(* Logix 5000 project; controller Drives_Line1 1756-L72 rev 20.13; software revision 20.04; part 12 of 21 *)
(* tags used below, declared in another part *)
   Bridle_02 : UDT_Bridle_2M;
   Bridle_03 : UDT_Bridle_2M;
   cu : UDT_Pinchroll;
   In_Commands : UDT_Commands;
   LineCmd : UDT_Commands_Line;
   LineCtrl : UDT_Control_Line;
   Out_Feedbacks : UDT_Fdbks;
   Out_Status : UDT_Status;
   TaskInterval_ms : DINT;
   TestConfig_Bridle_02a : UDT_Config_Bridle;
   TestConfig_Bridle_02b : UDT_Config_Bridle;
   TestConfig_cu : UDT_Config_Pinch;
   zConfigFromMaster : BOOL;
   zCuSpdTrimMltp : REAL;
   zPi : REAL;
   zSimulation : BOOL;
(* P15_Bridle_02, continued *)

ROUTINE R98_ToDrive   (* ladder *)
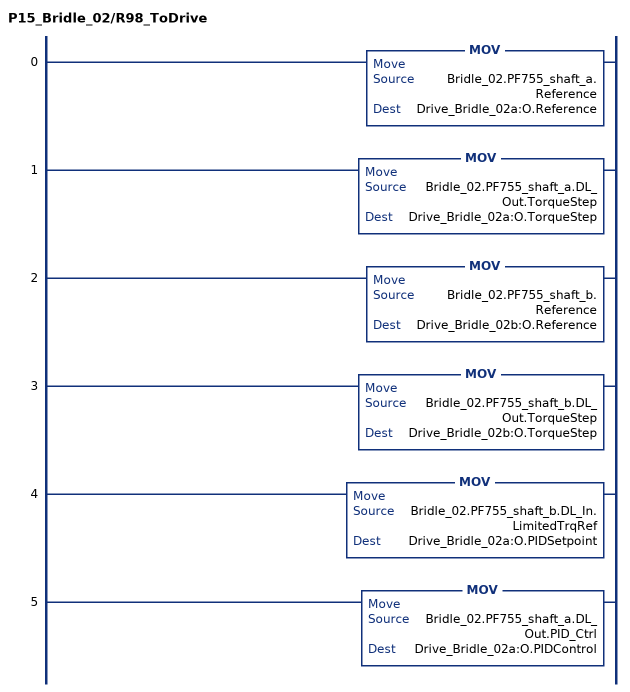
   0: MOV(Bridle_02.PF755_shaft_a.Reference,Drive_Bridle_02a:O.Reference);
   1: MOV(Bridle_02.PF755_shaft_a.DL_Out.TorqueStep,Drive_Bridle_02a:O.TorqueStep);
   2: MOV(Bridle_02.PF755_shaft_b.Reference,Drive_Bridle_02b:O.Reference);
   3: MOV(Bridle_02.PF755_shaft_b.DL_Out.TorqueStep,Drive_Bridle_02b:O.TorqueStep);
   4: MOV(Bridle_02.PF755_shaft_b.DL_In.LimitedTrqRef,Drive_Bridle_02a:O.PIDSetpoint);
   5: MOV(Bridle_02.PF755_shaft_a.DL_Out.PID_Ctrl,Drive_Bridle_02a:O.PIDControl);
END_ROUTINE

ROUTINE R999_Test   (* ladder *)
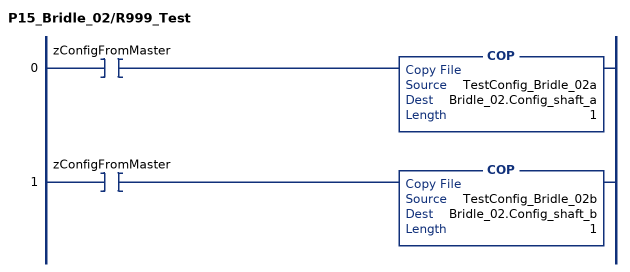
   0: XIC(zConfigFromMaster)COP(TestConfig_Bridle_02a,Bridle_02.Config_shaft_a,1);
   1: XIC(zConfigFromMaster)COP(TestConfig_Bridle_02b,Bridle_02.Config_shaft_b,1);
END_ROUTINE

ROUTINE R99_To_Master   (* ladder *)
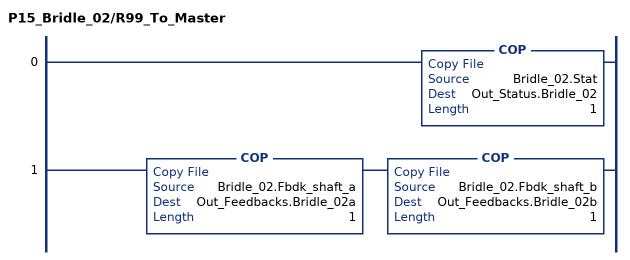
   0: COP(Bridle_02.Stat,Out_Status.Bridle_02,1);
   1: COP(Bridle_02.Fbdk_shaft_a,Out_Feedbacks.Bridle_02a,1)COP(Bridle_02.Fbdk_shaft_b,Out_Feedbacks.Bridle_02b,1);
END_ROUTINE
END_PROGRAM

PROGRAM P15b_rl_Cu   (* main routine R00_Main *)
VAR
   ADD_01 : FBD_MATH := (SourceB := 0.00068994303, Dest := 0.00068994303);
   aux1 : REAL;
   aux2 : REAL;
   BAND_01 : FBD_BOOLEAN_AND := (In3 := 1, In4 := 1, In5 := 1, In6 := 1, In7 := 1, In8 := 1);
   BAND_03 : FBD_BOOLEAN_AND := (In3 := 1, In4 := 1, In5 := 1, In6 := 1, In7 := 1, In8 := 1);
   BNOT_01 : FBD_BOOLEAN_NOT := (In := 1);
   BNOT_04 : FBD_BOOLEAN_NOT := (Out := 1);
   BNOT_06 : FBD_BOOLEAN_NOT := (Out := 1);
   cu2_Max_FBcounts : REAL := 5120.0;
   cu_FB_Count_Old : DINT;
   cu_FB_Diff : DINT;
   cu_FB_Update_Valid : BOOL;
   cu_Max_FBcounts : REAL := 5120.0;
   cu_RPMPerMPS : REAL := 5512.139;
   cu_SpdTrimMPS : REAL := 3.1769214e-06;
   cu_SpdTrimPct : REAL := 0.032127563;
   DIV_01 : FBD_MATH := (SourceA := 0.00053545943, SourceB := 100.0, Dest := 5.354594e-06);
   EQU_01 : FBD_COMPARE := (SourceA := 0.083333336);
   IO_State_cu : INT := 4;
   IO_State_Tmp_cu : INT := 16384;
   MUL_01 : FBD_MATH := (SourceA := 0.00068994303, SourceB := 5512.139, Dest := 3.803062);
   MUL_02 : FBD_MATH := (SourceA := 0.2);
   MUL_05 : FBD_MATH := (SourceA := 0.049963027, SourceB := 0.016666668, Dest := 0.00083271717);
   NEG_04 : FBD_MATH_ADVANCED := (Source := 0.233, Dest := -0.233);
   Ons : DINT := 1;
   PI_02 : PROP_INT := (In := 0.0045986176, Kp := 0.8, Wld := 0.1, HighLimit := 2.5, LowLimit := -2.5, ShapeKpPlus := 1.0, ShapeKpMinus := 1.0, ShapeWldPlus := 1.0, ShapeWldMinus := 1.0, RTSTime := 1, Out := 0.033255614, DeltaT := 0.05);
   PulsReset_PID : TIMER := (PRE := 250);
   RLIM_01 : RATE_LIMITER := (In := 0.00068994303, IncRate := 0.5, DecRate := 0.5, RTSTime := 1, Out := 0.00068994303, DeltaT := 0.05);
   SCL_09 : SCALE := (In := 0.1839509, InRawMax := 100.0, InRawMin := -100.0, InEUMax := 2.5, InEUMin := -2.5, Limiting := 1, Out := 0.0045986176);
   SCRV_01 : S_CURVE := (Initialize := 1, AbsAlgRamp := 1, AccelRate := 0.16, DecelRate := 0.16, JerkRate := 0.25, RTSTime := 1, DeltaT := 0.05);
   SSUM_03 : SELECTED_SUMMER := (In1 := 0.233, Gain1 := 1.0, In2 := -0.233, Gain2 := 1.0, Gain3 := 1.0, Select3 := 1, Gain4 := 1.0, Gain5 := 1.0, Gain6 := 1.0, Gain7 := 1.0, Gain8 := 1.0);
   SSUM_05 : SELECTED_SUMMER := (In1 := 0.00068994303, Gain1 := 1.0, Select1 := 1, Gain2 := 1.0, Gain3 := 1.0, Gain4 := 1.0, Gain5 := 1.0, Gain6 := 1.0, Gain7 := 1.0, Gain8 := 1.0, Out := 0.00068994303);
   SUB_02 : FBD_MATH := (SourceA := 6.741889, SourceB := 6.6660895, Dest := 0.075799465);
   TimeOn_PIDOn : TIMER := (PRE := 500);
   TofReset : TIMER := (PRE := 1000, ACC := 1000);
   TonNoResponse : TIMER[3] := ([0].PRE := 2500, [1].PRE := 2500, [2].PRE := 2500, [2].ACC := 2500, [2].EN := 1, [2].DN := 1);
   TonRefOn : TIMER := (PRE := 500);
   zcu_EncRes : DINT := 4096;
   zcu_Ki_SpdTrim : REAL := 0.1;
   zcu_Kp_SpdTrim : REAL := 0.8;
   zcu_Max_rev : DINT := 1500;
   zcu_MaxAccDec : REAL := 0.5;
   zcu_MaxTrimSpdTrim : REAL := 2.5;
   zcu_MinTrimSpdTrim : REAL := -2.5;
END_VAR

ROUTINE R00_Main   (* ladder *)
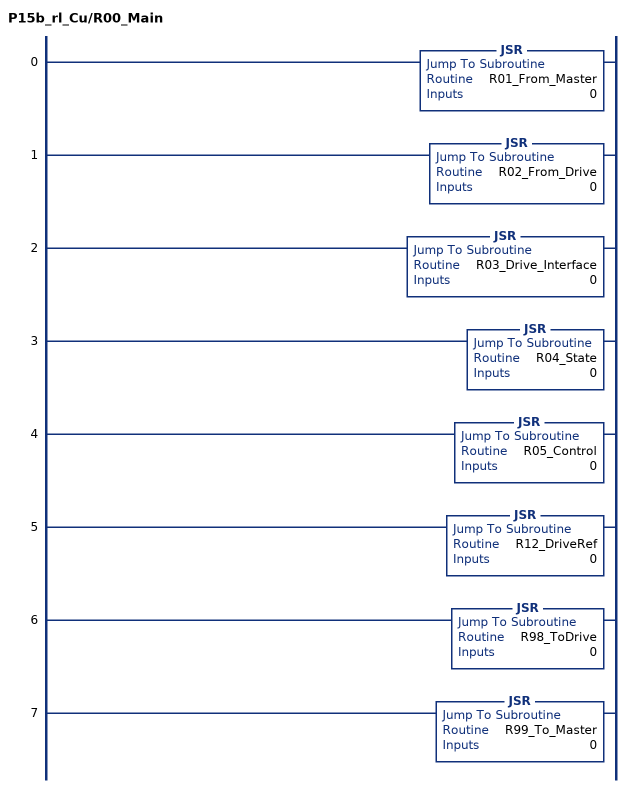
   0: JSR(R01_From_Master,0);
   1: JSR(R02_From_Drive,0);
   2: JSR(R03_Drive_Interface,0);
   3: JSR(R04_State,0);
   4: JSR(R05_Control,0);
   5: JSR(R12_DriveRef,0);
   6: JSR(R98_ToDrive,0);
   7: JSR(R99_To_Master,0);
END_ROUTINE

ROUTINE R01_From_Master   (* ladder *)
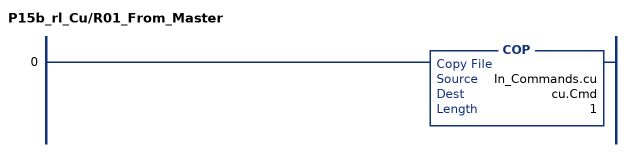
   0: COP(In_Commands.cu,cu.Cmd,1);
END_ROUTINE

ROUTINE R02_From_Drive   (* ladder *)
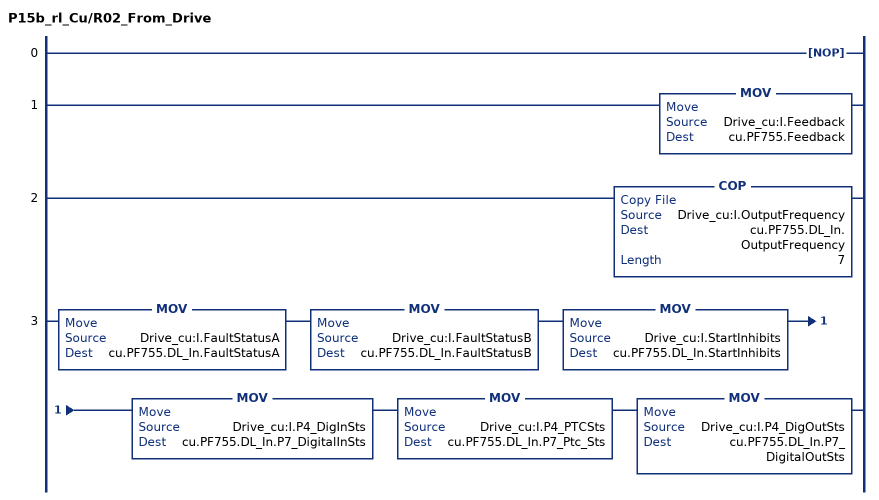
   0: NOP();
   1: MOV(Drive_cu:I.Feedback,cu.PF755.Feedback);
   2: COP(Drive_cu:I.OutputFrequency,cu.PF755.DL_In.OutputFrequency,7);
   3: MOV(Drive_cu:I.FaultStatusA,cu.PF755.DL_In.FaultStatusA)MOV(Drive_cu:I.FaultStatusB,cu.PF755.DL_In.FaultStatusB)MOV(Drive_cu:I.StartInhibits,cu.PF755.DL_In.StartInhibits)MOV(Drive_cu:I.P4_DigInSts,cu.PF755.DL_In.P7_DigitalInSts)MOV(Drive_cu:I.P4_PTCSts,cu.PF755.DL_In.P7_Ptc_Sts)MOV(Drive_cu:I.P4_DigOutSts,cu.PF755.DL_In.P7_DigitalOutSts);
END_ROUTINE

ROUTINE R03_Drive_Interface   (* ladder *)
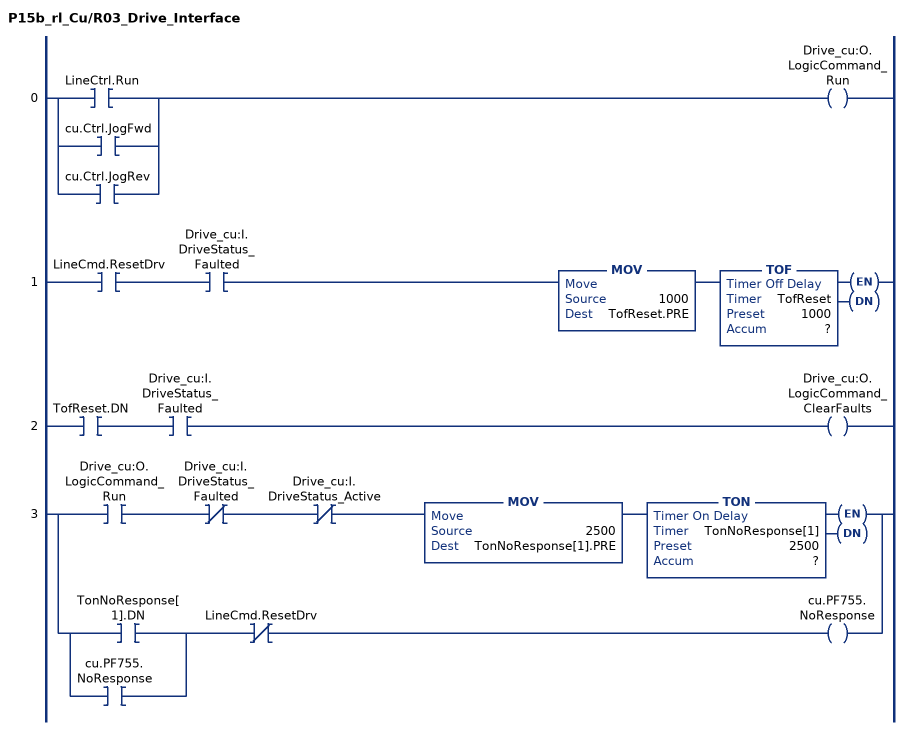
   0: [XIC(LineCtrl.Run) ,XIC(cu.Ctrl.JogFwd) ,XIC(cu.Ctrl.JogRev) ]OTE(Drive_cu:O.LogicCommand_Run);
   1: XIC(LineCmd.ResetDrv)XIC(Drive_cu:I.DriveStatus_Faulted)MOV(1000,TofReset.PRE)TOF(TofReset,?,?);
   2: XIC(TofReset.DN)XIC(Drive_cu:I.DriveStatus_Faulted)OTE(Drive_cu:O.LogicCommand_ClearFaults);
   3: [XIC(Drive_cu:O.LogicCommand_Run) XIO(Drive_cu:I.DriveStatus_Faulted) XIO(Drive_cu:I.DriveStatus_Active) MOV(2500,TonNoResponse[1].PRE) TON(TonNoResponse[1],?,?) ,[XIC(TonNoResponse[1].DN) ,XIC(cu.PF755.NoResponse) ] XIO(LineCmd.ResetDrv) OTE(cu.PF755.NoResponse) ];
END_ROUTINE

ROUTINE R04_State   (* ladder *)
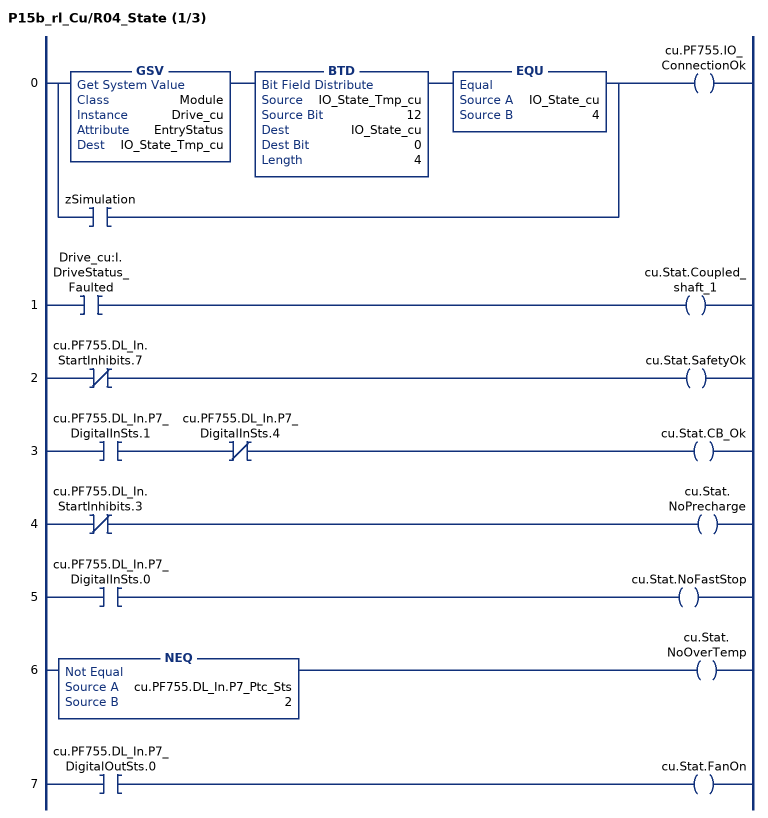
   0: [GSV(Module,Drive_cu,EntryStatus,IO_State_Tmp_cu) BTD(IO_State_Tmp_cu,12,IO_State_cu,0,4) EQU(IO_State_cu,4) ,XIC(zSimulation) ]OTE(cu.PF755.IO_ConnectionOk);
   1: XIC(Drive_cu:I.DriveStatus_Faulted)OTE(cu.Stat.Coupled_shaft_1);
   2: XIO(cu.PF755.DL_In.StartInhibits.7)OTE(cu.Stat.SafetyOk);
   3: XIC(cu.PF755.DL_In.P7_DigitalInSts.1)XIO(cu.PF755.DL_In.P7_DigitalInSts.4)OTE(cu.Stat.CB_Ok);
   4: XIO(cu.PF755.DL_In.StartInhibits.3)OTE(cu.Stat.NoPrecharge);
   5: XIC(cu.PF755.DL_In.P7_DigitalInSts.0)OTE(cu.Stat.NoFastStop);
   6: NEQ(cu.PF755.DL_In.P7_Ptc_Sts,2)OTE(cu.Stat.NoOverTemp);
   7: XIC(cu.PF755.DL_In.P7_DigitalOutSts.0)OTE(cu.Stat.FanOn);
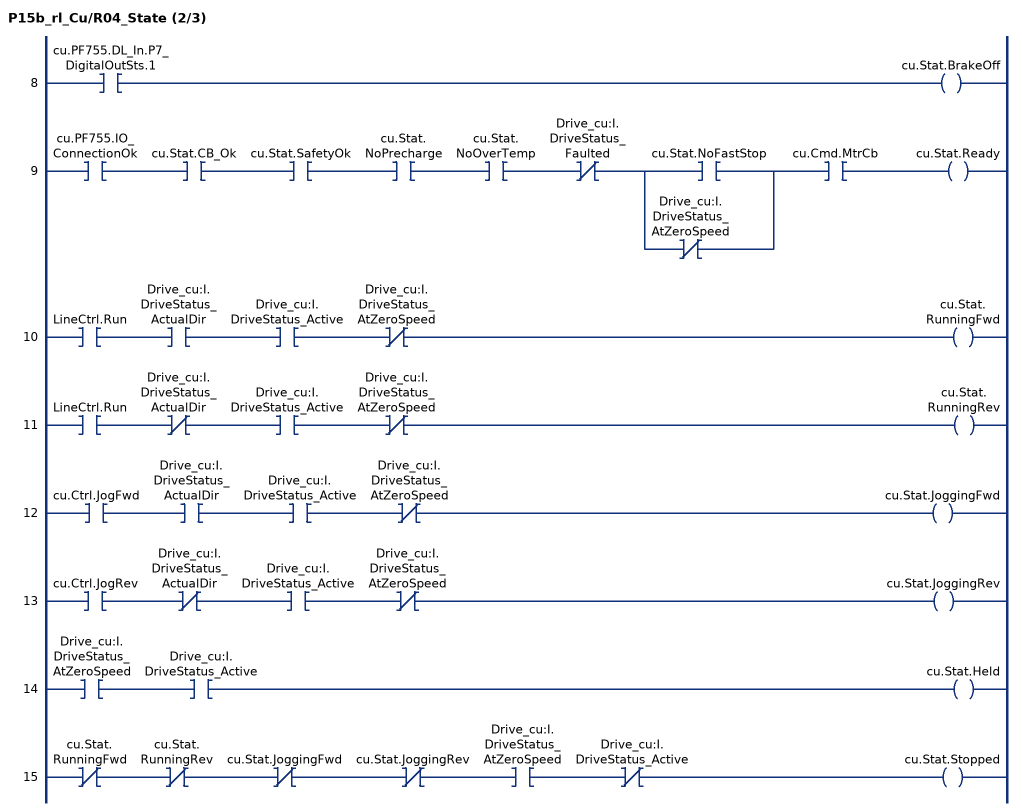
   8: XIC(cu.PF755.DL_In.P7_DigitalOutSts.1)OTE(cu.Stat.BrakeOff);
   9: XIC(cu.PF755.IO_ConnectionOk)XIC(cu.Stat.CB_Ok)XIC(cu.Stat.SafetyOk)XIC(cu.Stat.NoPrecharge)XIC(cu.Stat.NoOverTemp)XIO(Drive_cu:I.DriveStatus_Faulted)[XIC(cu.Stat.NoFastStop) ,XIO(Drive_cu:I.DriveStatus_AtZeroSpeed) ]XIC(cu.Cmd.MtrCb)OTE(cu.Stat.Ready);
   10: XIC(LineCtrl.Run)XIC(Drive_cu:I.DriveStatus_ActualDir)XIC(Drive_cu:I.DriveStatus_Active)XIO(Drive_cu:I.DriveStatus_AtZeroSpeed)OTE(cu.Stat.RunningFwd);
   11: XIC(LineCtrl.Run)XIO(Drive_cu:I.DriveStatus_ActualDir)XIC(Drive_cu:I.DriveStatus_Active)XIO(Drive_cu:I.DriveStatus_AtZeroSpeed)OTE(cu.Stat.RunningRev);
   12: XIC(cu.Ctrl.JogFwd)XIC(Drive_cu:I.DriveStatus_ActualDir)XIC(Drive_cu:I.DriveStatus_Active)XIO(Drive_cu:I.DriveStatus_AtZeroSpeed)OTE(cu.Stat.JoggingFwd);
   13: XIC(cu.Ctrl.JogRev)XIO(Drive_cu:I.DriveStatus_ActualDir)XIC(Drive_cu:I.DriveStatus_Active)XIO(Drive_cu:I.DriveStatus_AtZeroSpeed)OTE(cu.Stat.JoggingRev);
   14: XIC(Drive_cu:I.DriveStatus_AtZeroSpeed)XIC(Drive_cu:I.DriveStatus_Active)OTE(cu.Stat.Held);
   15: XIO(cu.Stat.RunningFwd)XIO(cu.Stat.RunningRev)XIO(cu.Stat.JoggingFwd)XIO(cu.Stat.JoggingRev)XIC(Drive_cu:I.DriveStatus_AtZeroSpeed)XIO(Drive_cu:I.DriveStatus_Active)OTE(cu.Stat.Stopped);
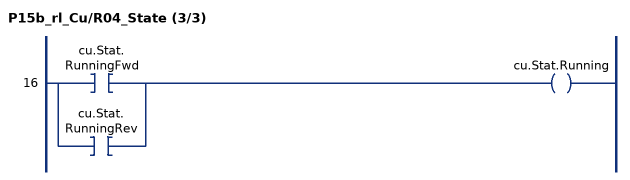
   16: [XIC(cu.Stat.RunningFwd) ,XIC(cu.Stat.RunningRev) ]OTE(cu.Stat.Running);
END_ROUTINE

ROUTINE R05_Control   (* ladder *)
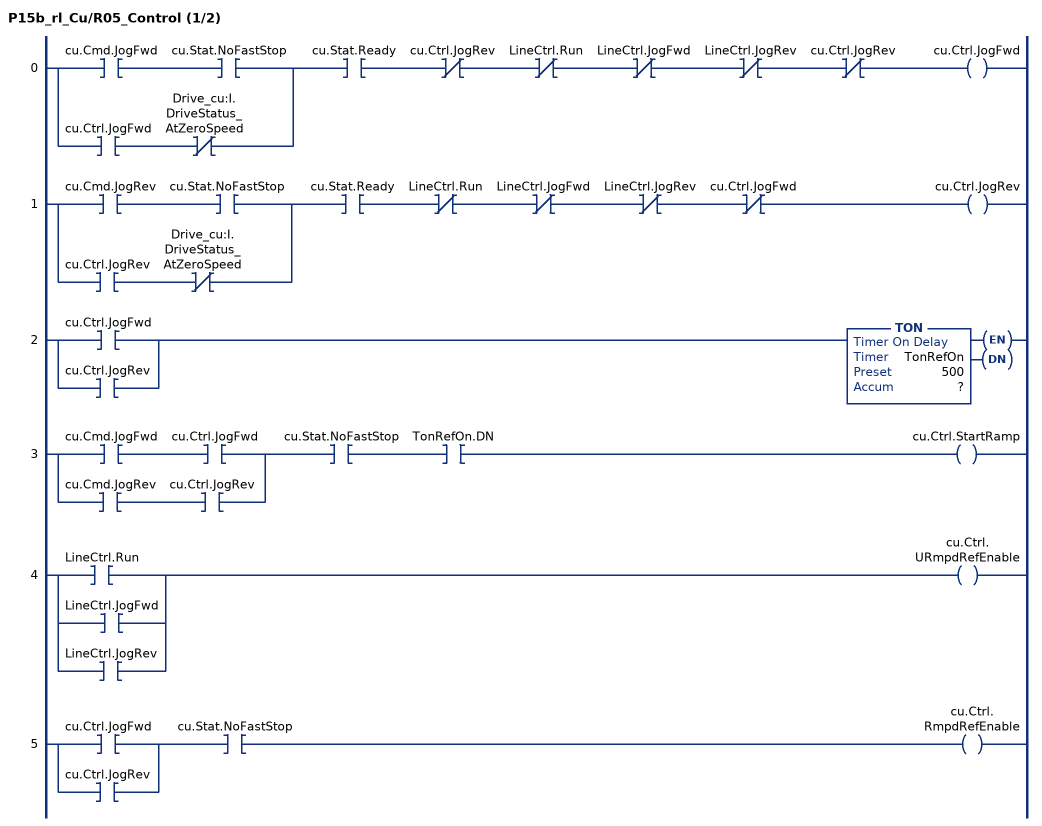
   0: [XIC(cu.Cmd.JogFwd) XIC(cu.Stat.NoFastStop) ,XIC(cu.Ctrl.JogFwd) XIO(Drive_cu:I.DriveStatus_AtZeroSpeed) ]XIC(cu.Stat.Ready)XIO(cu.Ctrl.JogRev)XIO(LineCtrl.Run)XIO(LineCtrl.JogFwd)XIO(LineCtrl.JogRev)XIO(cu.Ctrl.JogRev)OTE(cu.Ctrl.JogFwd);
   1: [XIC(cu.Cmd.JogRev) XIC(cu.Stat.NoFastStop) ,XIC(cu.Ctrl.JogRev) XIO(Drive_cu:I.DriveStatus_AtZeroSpeed) ]XIC(cu.Stat.Ready)XIO(LineCtrl.Run)XIO(LineCtrl.JogFwd)XIO(LineCtrl.JogRev)XIO(cu.Ctrl.JogFwd)OTE(cu.Ctrl.JogRev);
   2: [XIC(cu.Ctrl.JogFwd) ,XIC(cu.Ctrl.JogRev) ]TON(TonRefOn,?,?);
   3: [XIC(cu.Cmd.JogFwd) XIC(cu.Ctrl.JogFwd) ,XIC(cu.Cmd.JogRev) XIC(cu.Ctrl.JogRev) ]XIC(cu.Stat.NoFastStop)XIC(TonRefOn.DN)OTE(cu.Ctrl.StartRamp);
   4: [XIC(LineCtrl.Run) ,XIC(LineCtrl.JogFwd) ,XIC(LineCtrl.JogRev) ]OTE(cu.Ctrl.URmpdRefEnable);
   5: [XIC(cu.Ctrl.JogFwd) ,XIC(cu.Ctrl.JogRev) ]XIC(cu.Stat.NoFastStop)OTE(cu.Ctrl.RmpdRefEnable);
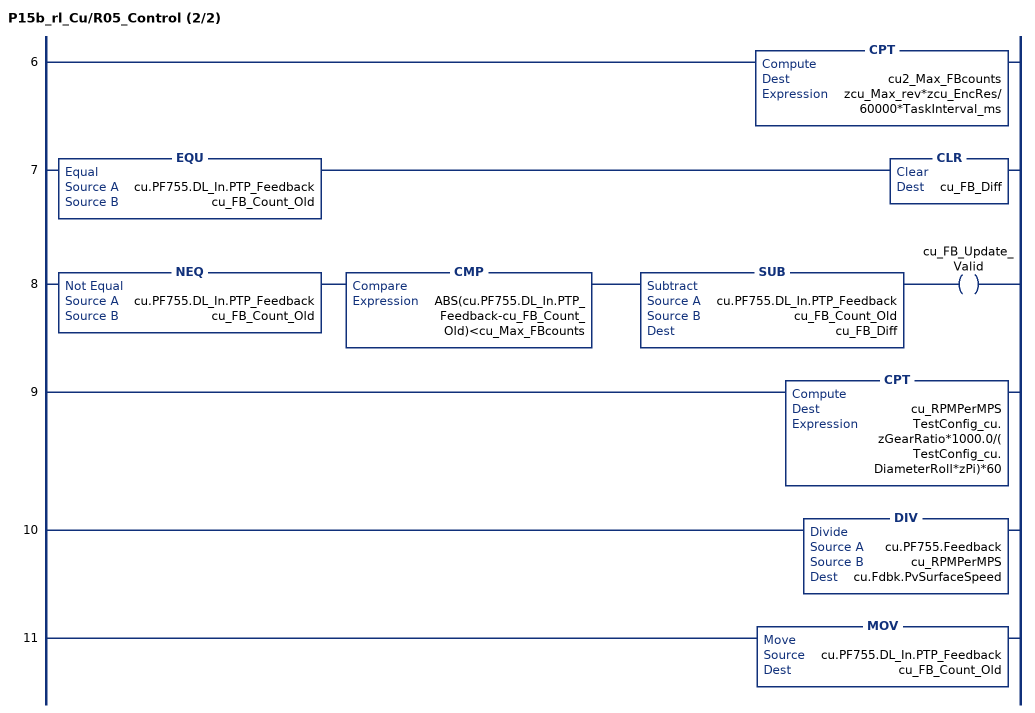
   6: CPT(cu2_Max_FBcounts,zcu_Max_rev*zcu_EncRes/60000*TaskInterval_ms);
   7: EQU(cu.PF755.DL_In.PTP_Feedback,cu_FB_Count_Old)CLR(cu_FB_Diff);
   8: NEQ(cu.PF755.DL_In.PTP_Feedback,cu_FB_Count_Old)CMP(ABS(cu.PF755.DL_In.PTP_Feedback-cu_FB_Count_Old)<cu_Max_FBcounts)SUB(cu.PF755.DL_In.PTP_Feedback,cu_FB_Count_Old,cu_FB_Diff)OTE(cu_FB_Update_Valid);
   9: CPT(cu_RPMPerMPS,TestConfig_cu.zGearRatio*1000.0/(TestConfig_cu.DiameterRoll*zPi)*60);
   10: DIV(cu.PF755.Feedback,cu_RPMPerMPS,cu.Fdbk.PvSurfaceSpeed);
   11: MOV(cu.PF755.DL_In.PTP_Feedback,cu_FB_Count_Old);
END_ROUTINE

ROUTINE R12_DriveRef   (* function block diagram *)
   SHEET 1   // Select jog speed reference
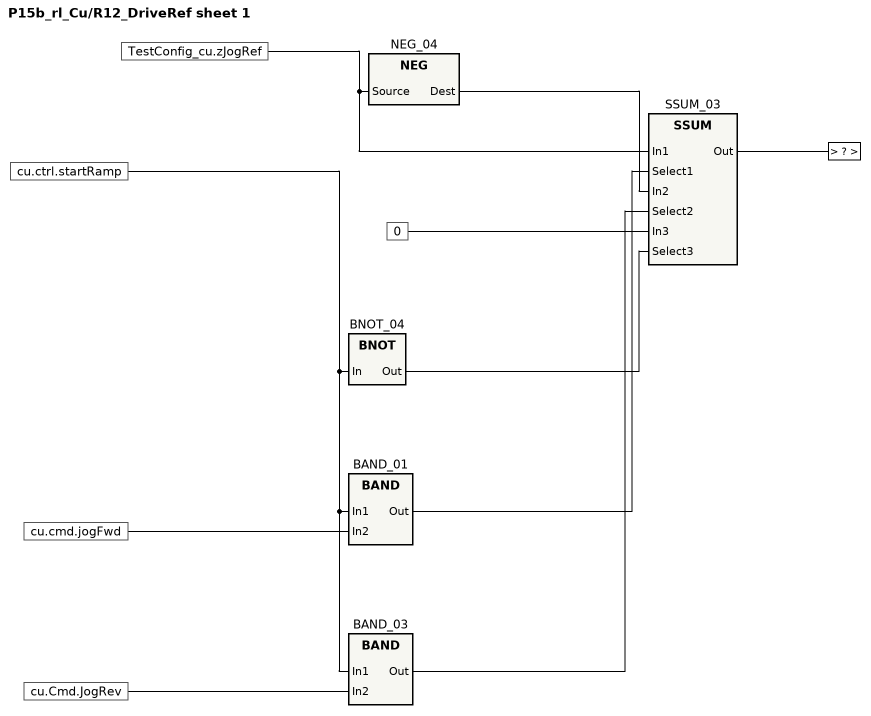
   BNOT_04 : BNOT(In := cu.ctrl.startRamp);
   BAND_01 : BAND(In1 := cu.ctrl.startRamp, In2 := cu.cmd.jogFwd);
   BAND_03 : BAND(In1 := cu.ctrl.startRamp, In2 := cu.Cmd.JogRev);
   NEG_04 : NEG(Source := TestConfig_cu.zJogRef);
   SSUM_03 : SSUM(In1 := TestConfig_cu.zJogRef, Select1 := BAND_01.Out, In2 := NEG_04.Dest, Select2 := BAND_03.Out, In3 := 0, Select3 := BNOT_04.Out);
   WIRE(?) := SSUM_03.Out;
   SHEET 2   // S-Curve
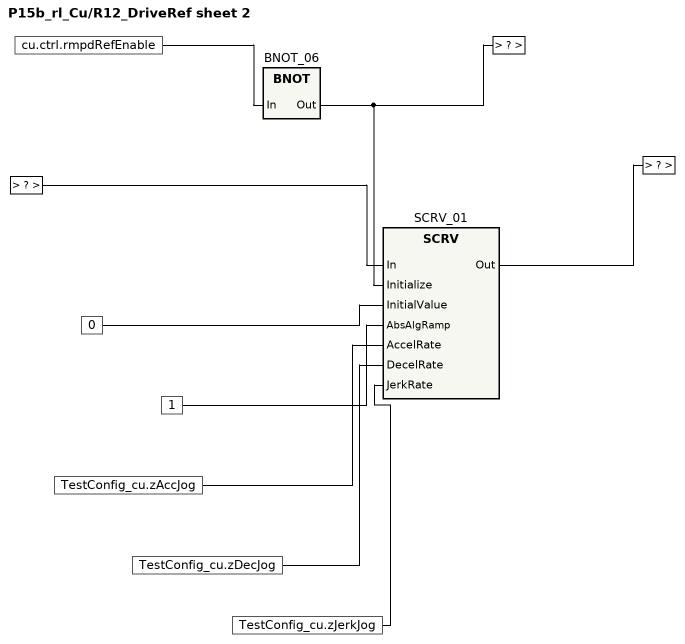
   BNOT_06 : BNOT(In := cu.ctrl.rmpdRefEnable);
   WIRE(?) := BNOT_06.Out;
   SCRV_01 : SCRV(In := WIRE(?), Initialize := BNOT_06.Out, InitialValue := 0, AbsAlgRamp := 1, AccelRate := TestConfig_cu.zAccJog, DecelRate := TestConfig_cu.zDecJog, JerkRate := TestConfig_cu.zJerkJog);
   WIRE(?) := SCRV_01.Out;
   SHEET 3   // Select ramped/unramped reference
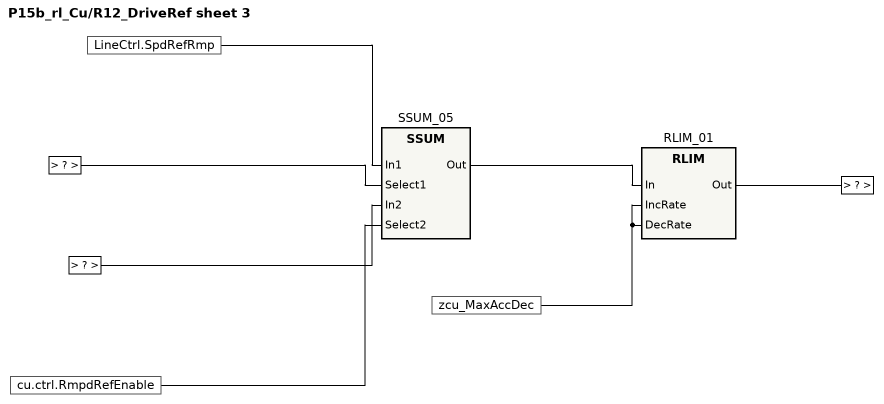
   SSUM_05 : SSUM(In1 := LineCtrl.SpdRefRmp, Select1 := WIRE(?), In2 := WIRE(?), Select2 := cu.ctrl.RmpdRefEnable);
   RLIM_01 : RLIM(In := SSUM_05.Out, IncRate := zcu_MaxAccDec, DecRate := zcu_MaxAccDec);
   WIRE(?) := RLIM_01.Out;
   SHEET 4   // Final speed reference
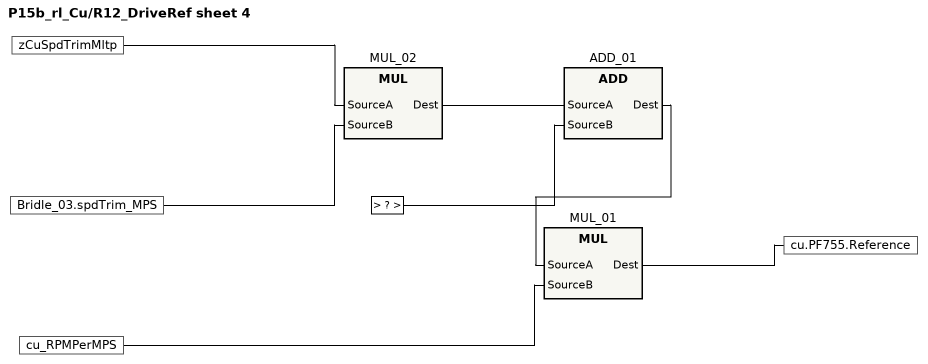
   MUL_02 : MUL(SourceA := zCuSpdTrimMltp, SourceB := Bridle_03.spdTrim_MPS);
   ADD_01 : ADD(SourceA := MUL_02.Dest, SourceB := WIRE(?));
   MUL_01 : MUL(SourceA := ADD_01.Dest, SourceB := cu_RPMPerMPS);
   cu.PF755.Reference := MUL_01.Dest;
END_ROUTINE

ROUTINE R98_ToDrive   (* ladder *)
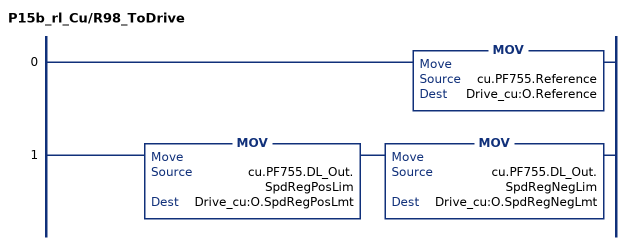
   0: MOV(cu.PF755.Reference,Drive_cu:O.Reference);
   1: MOV(cu.PF755.DL_Out.SpdRegPosLim,Drive_cu:O.SpdRegPosLmt)MOV(cu.PF755.DL_Out.SpdRegNegLim,Drive_cu:O.SpdRegNegLmt);
END_ROUTINE

ROUTINE R99_To_Master   (* ladder *)
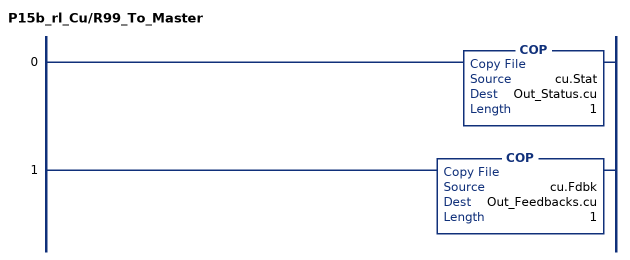
   0: COP(cu.Stat,Out_Status.cu,1);
   1: COP(cu.Fdbk,Out_Feedbacks.cu,1);
END_ROUTINE
END_PROGRAM
